// TIA Portal V20 export
DATA_BLOCK "DB_Contron_Coveyor_Belt"   // DB5
{ S7_Optimized_Access := 'TRUE' }
// stored: MemoryReserve 100
   VAR
      Pause_Conveyor_Belt_And_Carousel_Functional_Test : Bool;
   END_VAR
BEGIN
END_DATA_BLOCK
